{attribute 'enable_dynamic_creation'}
FUNCTION_BLOCK FutureCounterBlink EXTENDS FB_AbstructFuture
VAR_INPUT
END_VAR
VAR_OUTPUT
END_VAR
VAR
	_own_parameter: UINT;
	process_timer: TON;
	blink_timer: TON;
	_result :UDINT;
	_counter :UINT;
	_own_input: REFERENCE TO BOOL;
	_own_output: REFERENCE TO BOOL;
END_VAR

METHOD abort : BOOL
// The warning can be disabled here as the user is aware of the risk that the reference may not be valid by checking its validity
{warning disable C0371}
// Checking the VAR_IN_OUT reference, leave the current method in case of invalid reference
IF NOT __ISVALIDREF(_own_output) THEN
     RETURN;
END_IF

_own_output := FALSE;
abort := TRUE;

// The warning may be restored at the end of the access area
{warning restore C0371}
END_METHOD

PROPERTY counter : UINT
GET
counter := _counter;
END_GET
END_PROPERTY

METHOD execute : BOOL
VAR_INPUT
END_VAR
VAR_INST
	input_memory :BOOL;
END_VAR
// The warning can be disabled here as the user is aware of the risk that the reference may not be valid by checking its validity
{warning disable C0371}
// Checking the VAR_IN_OUT reference, leave the current method in case of invalid reference
IF NOT __ISVALIDREF(_own_output) OR NOT __ISVALIDREF(_own_input) THEN
     RETURN;
END_IF

_own_output := TRUE;
IF _own_input AND NOT input_memory THEN
	_counter := counter + 1;
END_IF
input_memory := _own_input;
IF _counter > _own_parameter THEN
	execute := TRUE;
END_IF

// The warning may be restored at the end of the access area
{warning restore C0371}
END_METHOD

METHOD init : BOOL
VAR_INPUT
END_VAR
// The warning can be disabled here as the user is aware of the risk that the reference may not be valid by checking its validity
{warning disable C0371}
// Checking the VAR_IN_OUT reference, leave the current method in case of invalid reference
IF NOT __ISVALIDREF(_own_output) THEN
	_result := 1;
     RETURN;
END_IF

_own_output := FALSE;
process_timer(IN := FALSE);
blink_timer(IN := FALSE);
_counter := 0;
init := TRUE;

// The warning may be restored at the end of the access area
{warning restore C0371}
END_METHOD

PROPERTY input : REFERENCE TO BOOL;
SET
_own_input REF= input;
END_SET
END_PROPERTY

PROPERTY nErrorID : UDINT
GET
nErrorID := _result;
END_GET
END_PROPERTY

PROPERTY output : REFERENCE TO BOOL;
SET
_own_output REF= output;
END_SET
END_PROPERTY

PROPERTY own_parameter : UINT
GET
own_parameter := _own_parameter;
END_GET
SET
_own_parameter := own_parameter;
END_SET
END_PROPERTY

METHOD quit : BOOL
THIS^.init();
quit := TRUE;
END_METHOD

END_FUNCTION_BLOCK

(* stored: Version 1.1.0.1, ProductVersion 3.1.4024.12
   POU FutureCounterBlink: Id {fcedd839-491a-4b82-962e-a6b212add423}, SpecialFunc None
   Method abort: Id {0318e039-5936-41e7-9acc-72e5c11c7579}
   Property counter: Id {d21e7cd7-0ef0-4123-a4e3-71fe9855b00a}
   Get Get: Id {a2a1935b-4339-4663-9b2a-10527d776baa}
   Method execute: Id {06ca504b-2230-462e-b402-b0513637b891}
   Method init: Id {0506fa37-b033-4ecf-a1b9-39ffd68590c2}
   Property input: Id {9b9ce6d4-2b7c-46f1-863a-ec0e0ee528c8}
   Set Set: Id {394f91d6-bbd4-402b-9daf-3e63549cb838}
   Property nErrorID: Id {16e63a23-0f02-402f-9998-37a3e09307d6}
   Get Get: Id {10902b3b-ec3f-43fc-b121-362377561d1c}
   Property output: Id {b3cff984-3339-47bc-bc72-9fee666901a0}
   Set Set: Id {cc76f589-3252-467a-a02f-9f4006b5aa11}
   Property own_parameter: Id {44c22855-b665-42b9-9698-003553798c6b}
   Get Get: Id {a4ce69b5-d711-41f1-b7ea-5a7f1940c7a1}
   Set Set: Id {20314786-f00f-435f-bd37-c1bd1124cdd5}
   Method quit: Id {77d78392-ba97-4c0d-a7ef-71aa64534b7c} *)
